(* IEC 61131-3 sources: ICARU_FB_v2/icarufb-dut-code/stcompiler, 15 files *)

(* ---- CAR_SEMAPHORE.st ---- *)
(* Generated by xml2st *)
FUNCTION_BLOCK CAR_SEMAPHORE
  EVENT_INPUT
    INIT;
    REQ;
    RECONF;
  END_EVENT
  EVENT_OUTPUT
    INITO;
    CNF;
    RECONFO;
  END_EVENT

  EC_STATES
    START;
    INIT: INIT -> INITO;
    REQ: ALG_REQ -> CNF;
    RECONF: -> CNF, ALG_RECONF -> RECONFO;
  END_STATES

  EC_TRANSITIONS
    INIT TO START := 1;
    START TO REQ := REQ;
    START TO INIT := INIT;
    REQ TO START := 1;
    START TO RECONF := RECONF;
  END_TRANSITIONS

  VAR_INPUT
    CYCLE: BYTE;
  END_VAR

  VAR_OUTPUT
    RED: BOOL;
    YELLOW: BOOL;
    GREEN: BOOL;
  END_VAR

  ALGORITHM INIT IN ST:
RED := TRUE;
GREEN := FALSE;
YELLOW := FALSE;
  END_ALGORITHM

  ALGORITHM ALG_REQ IN ST:
RED := FALSE;
YELLOW := FALSE;
GREEN := FALSE;
IF(CYCLE = 0) THEN
 RED:=TRUE;
END_IF;
IF(CYCLE=1)THEN
 GREEN:=TRUE;
END_IF;
IF(CYCLE=2)THEN
 YELLOW:=TRUE;
END_IF;
  END_ALGORITHM

  ALGORITHM ALG_RECONF IN ST:
RED:=FALSE;
YELLOW:=TRUE;
GREEN:=FALSE;
  END_ALGORITHM

END_FUNCTION_BLOCK

(* ---- E_SPLIT.st ---- *)
(* Generated by xml2st *)
FUNCTION_BLOCK E_SPLIT
  EVENT_INPUT
    EI1;
  END_EVENT
  EVENT_OUTPUT
    EO1;
    EO2;
  END_EVENT

  EC_STATES
    RUN: -> EO1, -> EO2;
    START;
  END_STATES

  EC_TRANSITIONS
    START TO RUN := EI1;
    RUN TO START := 1;
  END_TRANSITIONS

  VAR_INPUT
  END_VAR

  VAR_OUTPUT
  END_VAR

END_FUNCTION_BLOCK

(* ---- fb_flash.st ---- *)
FUNCTION_BLOCK FLASHER
	EVENT_INPUT
		FLASH;
	END_EVENT
	EVENT_OUTPUT
		Q;
	END_EVENT

	EC_STATES
		START; (* Initial state *)
		ST_FLASH: ALG_FLASH -> Q;
	END_STATES

	EC_TRANSITIONS
		START TO ST_FLASH := FLASH;
		ST_FLASH TO START := 1;
	END_TRANSITIONS

	VAR_OUTPUT
		LED: BOOL;
	END_VAR

	ALGORITHM ALG_FLASH IN ST:
		LED := NOT LED;
	END_ALGORITHM

END_FUNCTION_BLOCK

(* ---- fb_io_reader.st ---- *)
FUNCTION_BLOCK IO_READER
	EVENT_INPUT
		INIT;
		RSP;
	END_EVENT

	EVENT_OUTPUT
		INIT0;
		IND;
	END_EVENT

	EC_STATES
		START; (* Initial state *)
		INIT: ALG_INIT -> INIT0;
		READ: ALG_READ -> IND;
	END_STATES

	EC_TRANSITIONS
		START TO INIT := INIT;
		INIT TO START := 1;
		START TO READ := RSP;
		READ TO START := 1;
	END_TRANSITIONS

	VAR_INPUT
		QI: BOOL;
		PARAMS: INT;
		SD_1: INT; (* Address *)
	END_VAR

	VAR_OUTPUT
		QO: BOOL;
		STATUS: INT;
		RD_1: INT;
	END_VAR

	ALGORITHM ALG_READ IN ST:
		RD_1 := GET_REG(SD_1);
	END_ALGORITHM
	ALGORITHM ALG_INIT IN ST:

	END_ALGORITHM
END_FUNCTION_BLOCK

(* ---- fb_io_writer.st ---- *)
FUNCTION_BLOCK IO_WRITER
	EVENT_INPUT
		INIT;
		REQ;
	END_EVENT

	EVENT_OUTPUT
		INIT0;
		CNF;
	END_EVENT

	EC_STATES
		START; (* Initial state *)
		INIT: ALG_INIT -> INIT0;
		WRITE: ALG_WRITE->CNF;
	END_STATES

	EC_TRANSITIONS
		START TO INIT  := INIT;
		START TO WRITE := REQ;
		WRITE TO START := 1;
		INIT TO START  := 1;
	END_TRANSITIONS

	VAR_INPUT
		QI: BOOL;
		PARAMS: INT;
		SD_1: INT; (* Address *)
		SD_2: INT; (* Value *)
	END_VAR

	VAR_OUTPUT
		QO: BOOL;
		STATUS: INT;
		RD_1: INT;
	END_VAR

	ALGORITHM ALG_WRITE IN ST:
		SET_REG(SD_1, SD_2);
	END_ALGORITHM
	ALGORITHM ALG_INIT IN ST:

	END_ALGORITHM
END_FUNCTION_BLOCK

(* ---- fb_publisher.st ---- *)
FUNCTION_BLOCK PUBLISHER
	EVENT_INPUT
		INIT;
		REQ;
	END_EVENT

	EVENT_OUTPUT
		INIT0;
		CNF;
	END_EVENT

	EC_STATES

		INIT: ALG_INIT -> INIT0;
		START; (* Initial state *)
	END_STATES

	EC_TRANSITIONS
		START TO INIT := INIT;

	END_TRANSITIONS

	VAR_INPUT
		Q1: BOOL;
		PARAMS: INT; (* Address *)
		SD_1: INT;
	END_VAR

	VAR_OUTPUT
		QO: BOOL;
		STATUS: INT;
	END_VAR

	ALGORITHM READ IN ST:

	END_ALGORITHM
	ALGORITHM ALG_INIT IN ST:

	END_ALGORITHM
END_FUNCTION_BLOCK

(* ---- fb_subscriber.st ---- *)
FUNCTION_BLOCK SUBSCRIBER
	EVENT_INPUT
		INIT;
		RSP;
	END_EVENT

	EVENT_OUTPUT
		INIT0;
		IND;
	END_EVENT

	EC_STATES
		START; (* Initial state *)
		INIT: ALG_INIT -> INIT0;

	END_STATES

	EC_TRANSITIONS
		START TO INIT := INIT;

	END_TRANSITIONS

	VAR_INPUT
		Q1: BOOL;
		PARAMS: INT; (* Address *)
		SD_1: INT;
	END_VAR

	VAR_OUTPUT
		QO: BOOL;
		STATUS: INT;
		RD_1: INT; (* Value *)
	END_VAR

	ALGORITHM READ IN ST:

	END_ALGORITHM
	ALGORITHM ALG_INIT IN ST:

	END_ALGORITHM
END_FUNCTION_BLOCK

(* ---- fb_tmp_control.st ---- *)
FUNCTION_BLOCK TMP_CONTROL
  EVENT_INPUT
  	INIT;
  	READ;
  END_EVENT
  EVENT_OUTPUT
  	INITO;
  	Q;
  END_EVENT

  EC_STATES
    START; (* Initial state *)
    ST_INIT: ALG_INIT -> INITO;
    ST_READ: ALG_READ -> Q;
  END_STATES

  EC_TRANSITIONS
    START TO ST_INIT := INIT;
    ST_INIT TO START := 1;
    START TO ST_READ := READ;
    ST_READ TO START := 1;
  END_TRANSITIONS

  VAR_INPUT
    TEMP: REAL;
  END_VAR
  VAR_OUTPUT
    REF: BOOL;
  END_VAR

  ALGORITHM ALG_INIT IN ST:
    REF := FALSE;
  END_ALGORITHM

  ALGORITHM ALG_READ IN ST:
    IF TEMP > 30.0 THEN
      REF := TRUE;
    END_IF ;
	IF TEMP < 20.0 THEN
      REF := FALSE;
    END_IF;
  END_ALGORITHM

END_FUNCTION_BLOCK

FUNCTION_BLOCK TMP_CONTROL3
	EVENT_INPUT
		INIT;
		ACT;
	END_EVENT

	EVENT_OUTPUT
		R;
	END_EVENT

	EC_STATES
		START; (* Initial state *)
		INIT: ALG_INIT -> R;
		PROC: TMPCTL -> R;
	END_STATES

	EC_TRANSITIONS
		START TO INIT := INIT AND ACT;
		INIT TO START := 1;
		START TO PROC := ACT;
		PROC TO START := 1;
	END_TRANSITIONS

	VAR_INPUT
		TMP: REAL;
	END_VAR

	VAR_OUTPUT
		Q: BOOL;
		OT:INT;
	END_VAR

	VAR
		Va : INT := 10;
	END_VAR

	ALGORITHM TMPCTL IN ST:

		IF Q = 63 OR Q = 78 THEN
			OT := 100;
			Q:= TRUE;
		END_IF;
		IF TMP < 5 THEN
			Q:= FALSE;
		END_IF;

	END_ALGORITHM
	ALGORITHM ALG_INIT IN ST:
		Q := FALSE;
	END_ALGORITHM
END_FUNCTION_BLOCK

FUNCTION_BLOCK TMP_CONTROL2
	EVENT_INPUT
		INIT;
		ACT;
	END_EVENT

	EVENT_OUTPUT
		R;
	END_EVENT

	EC_STATES
		START; (* Initial state *)
		INIT: ALG_INIT -> R;
		PROC: TMPCTL -> R;
	END_STATES

	EC_TRANSITIONS
		START TO INIT := INIT AND ACT;
		INIT TO START := 1;

	END_TRANSITIONS

	VAR_INPUT
		TMP: INT;
	END_VAR

	VAR_OUTPUT
		Q: BOOL;
	END_VAR

	VAR
		V1 : BOOL:= 10;
	END_VAR

	ALGORITHM TMPCTL IN ST:

		TMP := 10;

	END_ALGORITHM
	ALGORITHM ALG_INIT IN ST:
		Q := FALSE;
	END_ALGORITHM
END_FUNCTION_BLOCK

(* ---- PUB_2.st ---- *)
(* Generated by xml2st *)
FUNCTION_BLOCK PUB_2
  EVENT_INPUT
    INIT;
    REQ;
  END_EVENT
  EVENT_OUTPUT
    INIT0;
  END_EVENT

  EC_STATES
    START;
    SEND: ALG_SND ->;
    INIT: ALG_INIT -> INIT0;
  END_STATES

  EC_TRANSITIONS
    START TO INIT := INIT;
    START TO SEND := REQ;
    SEND TO START := 1;
    INIT TO START := 1;
  END_TRANSITIONS

  VAR_INPUT
    ID: INT;
    RD_1: INT;
    RD_2: BOOL;
  END_VAR

  VAR_OUTPUT
  END_VAR

  VAR
    RD_1_: INT;
    RD_2_: BOOL;
  END_VAR

  ALGORITHM ALG_SND IN ST:
   (* IF (NOT(RD_1_ = RD_1)) OR (NOT(RD_2_ = RD_2)) THEN *)
      ASM
		LOAD RD_1_
		LOAD RD_1
		IFEQ GOTO +2
		GOTO send
		LOAD RD_2_
		LOAD RD_2
		IFEQ GOTO endif
		send:
	    LOAD RD_1
	    LOAD RD_2
	    CONST 2
	    LOAD ID
	    NISND

		LOAD RD_1
		STORE RD_1_
		LOAD RD_2
		STORE RD_2_
		endif:
	  END_ASM
	(*  RD_1_ := RD_1;
	  RD_2_ := RD_2;
	END_IF;*)
  END_ALGORITHM

  ALGORITHM ALG_INIT IN ST:

  END_ALGORITHM

END_FUNCTION_BLOCK

(* ---- SEM_CONTROL.st ---- *)
(* Generated by xml2st *)
FUNCTION_BLOCK SEM_CONTROL
  EVENT_INPUT
    INIT;
    ETIME;
  END_EVENT
  EVENT_OUTPUT
    INIT0;
    SET_SEMAPHORE;
  END_EVENT

  EC_STATES
    RUN: ALG_RUN -> SET_SEMAPHORE;
    START;
    INIT;
  END_STATES

  EC_TRANSITIONS
    START TO INIT := INIT;
    START TO RUN := ETIME;
    INIT TO START := 1;
    RUN TO START := 1;
  END_TRANSITIONS

  VAR_INPUT
    R: REAL;
  END_VAR

  VAR_OUTPUT
    SEMAPHORE_1: BYTE;
    SEMAPHORE_2: BYTE;
    SEMAPHORE_3: BYTE;
    SEMAPHORE_4: BYTE;
  END_VAR

  ALGORITHM ALG_INIT IN ST:
SEMAPHORE_1 := 0; SEMAPHORE_2 := 0; SEMAPHORE_3 := 0; SEMAPHORE_4 := 0;
  END_ALGORITHM

  ALGORITHM ALG_RUN IN ST:
 IF(SEMAPHORE_2 = 0) THEN  SEMAPHORE_1 := SEMAPHORE_1 + 1;  IF(SEMAPHORE_1 >= 3) THEN   SEMAPHORE_1 := 0;   SEMAPHORE_2 := 1;  END_IF; ELSE  SEMAPHORE_2 := SEMAPHORE_2 + 1;  IF(SEMAPHORE_2 >= 3) THEN   SEMAPHORE_1 := 1;   SEMAPHORE_2 := 0;  END_IF;  END_IF; R:=2.3 + 4.5; R:=(R+1.2)*3.0; R := R/2.0;
  END_ALGORITHM

END_FUNCTION_BLOCK

(* ---- SUB_2.st ---- *)
(* Generated by xml2st *)
FUNCTION_BLOCK SUB_2
  EVENT_INPUT
    INIT;
  END_EVENT
  EVENT_OUTPUT
    INIT0;
    RSP;
  END_EVENT

  EC_STATES
    START;
    RCV: ALG_RCV -> RSP;
    INIT: ALG_INIT -> INIT0;
  END_STATES

  EC_TRANSITIONS
    START TO INIT := INIT;
    INIT TO START := 1;
    START TO RCV := 1;
    RCV TO START := 1;
  END_TRANSITIONS

  VAR_INPUT
    ID: BOOL;
  END_VAR

  VAR_OUTPUT
    SD_1: INT;
    SD_2: BOOL;
  END_VAR

  ALGORITHM ALG_RCV IN ST:
ASM
    CONST 2
	LOAD ID
	NIRCV
	IF GOTO process
	GOTO out
process:
	STORE SD_1
	STORE SD_2
out:
	END_ASM
  END_ALGORITHM

  ALGORITHM ALG_INIT IN ST:

  END_ALGORITHM

END_FUNCTION_BLOCK

(* ---- SWITCHER.st ---- *)
(* Generated by xml2st *)
FUNCTION_BLOCK SWITCHER
  EVENT_INPUT
    INIT;
    REQ;
  END_EVENT
  EVENT_OUTPUT
    INITO;
    CNF;
  END_EVENT

  EC_STATES
    START;
    INIT: INIT -> INITO;
    REQ: REQ -> CNF;
  END_STATES

  EC_TRANSITIONS
    INIT TO START := 1;
    START TO REQ := REQ;
    START TO INIT := INIT;
    REQ TO START := 1;
  END_TRANSITIONS

  VAR_INPUT
    SIGIN: BOOL;
  END_VAR

  VAR_OUTPUT
    PIN: BYTE;
    VAL: BOOL;
    COUNT: BYTE;
  END_VAR

  ALGORITHM INIT IN ST:
COUNT:=0;
VAL:=0;
  END_ALGORITHM

  ALGORITHM REQ IN ST:
IF SIGIN THEN
  COUNT := COUNT + 1;
  IF (COUNT > 3) THEN
    COUNT := 0;
    VAL := NOT VAL;
  END_IF;
  PIN := 200 + COUNT;
END_IF;
  END_ALGORITHM

END_FUNCTION_BLOCK

(* ---- E_CYCLE.st ---- *)
CUSTOM FUNCTION_BLOCK E_DELAY
	EVENT_INPUT
		START;
		STOP;
	END_EVENT

	EVENT_OUTPUT
		EO;
	END_EVENT

	VAR_INPUT
		DT:INT;
	END_VAR

	VAR
		oldt: INT;
		count:INT;
		state: INT;
	END_VAR

	ALGORITHM ALG_INIT:
		oldt := GET_REG(100);
		count := 0;
		state := 0;
	END_ALGORITHM
	ALGORITHM ALG_RUN:
		IF(START) THEN
			state :=1;
			START := 0;
			count := 0;
			oldt := GET_REG(100);
		END_IF;
		IF(STOP)THEN
			state := 0;
			EO := 0;
		END_IF;
		IF(EO) THEN
			EO := 0;
		END_IF;
		IF(state = 1) THEN
			IF(NOT (oldt = GET_REG(100))) THEN
				count := count + 1;
				IF(count = DT) THEN
					EO := 1;
					count := 0;
				END_IF;
				oldt := GET_REG(100);
			END_IF;
		END_IF;
	END_ALGORITHM

END_FUNCTION_BLOCK

(* ---- E_DELAY.st ---- *)
CUSTOM FUNCTION_BLOCK E_DELAY
	EVENT_INPUT
		START;
		STOP;
	END_EVENT

	EVENT_OUTPUT
		EO;
	END_EVENT

	VAR_INPUT
		DT:BYTE;
	END_VAR

	VAR
		oldt: BYTE;
		count:BYTE;
		state: BYTE;
	END_VAR

	ALGORITHM ALG_INIT:
		oldt := GET_REG(100);
		count := 0;
		state := 0;
	END_ALGORITHM
	ALGORITHM ALG_RUN:
		IF(START) THEN
			state :=1;
			START := 0;
			count := GET_REG(100);
		END_IF;

		IF(state = 1) THEN
			IF(NOT (oldt = GET_REG(100))) THEN
				count := count + 1;
				IF(count = DT) THEN
					EO := 1;
					state := 0;
				END_IF;
				oldt := GET_REG(100);

			END_IF;
		END_IF;

		count := 2 + 4.5;
	END_ALGORITHM

END_FUNCTION_BLOCK

(* ---- E_TEST.st ---- *)
CUSTOM FUNCTION_BLOCK E_TEST
	EVENT_INPUT
		START;
	END_EVENT

	EVENT_OUTPUT
		EO;
	END_EVENT

	VAR_INPUT
		DT:BYTE;
	END_VAR

	VAR
		num:REAL;
	END_VAR

	ALGORITHM ALG_INIT:
		num := 2.4;
	END_ALGORITHM
	ALGORITHM ALG_RUN:
		num:=num + 3.5;
	END_ALGORITHM

END_FUNCTION_BLOCK
